// TIA Portal V19 export
TYPE "LEXCHANGETRAY_typeRoller_toLogisticsRecieve"
// stored: Access Published
   STRUCT
      feedback : "LEXCHANGETRAY_typeLogistics_toRollerFeedback";
      req : "LEXCHANGETRAY_typeLogistics_toRollerReq";
   END_STRUCT;
END_TYPE
